// TwinCAT 3 PLC project Untitled1
// ProgramVersion: 3.1.4023.0
// libraries:
//   Tc2_Standard, * (Beckhoff Automation GmbH)
//   Tc2_System, * (Beckhoff Automation GmbH)
//   Tc2_Utilities, * (Beckhoff Automation GmbH)
//   Tc3_Module, * (Beckhoff Automation GmbH)
// project tree:
//   DUTs/BundleData/ Bundle.TcDUT (not stored), Interval.TcDUT (not stored), Material.TcDUT, PositionMaterials.TcDUT (not stored)
//   DUTs/Conveyors/ Conveyor.TcPOU, ConveyorLSC.TcPOU (not stored), ConveyorMode.TcDUT (not stored), ConveyorSC.TcPOU, ConveyorSC_NC.TcPOU
//   DUTs/ SectionTask.TcDUT, Surface.TcDUT
//   GVLs/ CONSTS.TcGVL
//   HARDWARE_DISTRUBUTION/ ConveyorSyncUnit.TcPOU
//   / PlcTask.TcTTO
//   POUs/Helper Functions/ BundleIsValid.TcPOU (not stored)
//   POUs/ IndexedBuffer.TcPOU, Junction.TcPOU, MAIN.TcPOU
// real-time tasks:
//   TASK PlcTask: cycle T#10ms, priority 20, ADS port 350

CONFIGURATION Untitled1
    RESOURCE PLC ON TwinCAT3
        TASK PlcTask(INTERVAL := T#10ms, PRIORITY := 20);
        PROGRAM MAIN WITH PlcTask : MAIN;
    END_RESOURCE
END_CONFIGURATION

// ---- DUTs/BundleData/Material.TcDUT
TYPE Material :
STRUCT
	code : STRING;
	width : LREAL;
	length : LREAL;
END_STRUCT
END_TYPE
(*
use this struct to keep track of where materials are
materials enter the system when pulled from their magazine/skid and exit the system when placed on the bundle or otherwise lost
*)

// ---- DUTs/SectionTask.TcDUT
{attribute 'qualified_only'}
//{attribute 'strict'}
TYPE SectionTask :
(
	IDLE,
	ALIGN,
	ACTIVE,
	DISCHARGE,
	COMPLETE,
	
	size
);
END_TYPE

// ---- DUTs/Surface.TcDUT
{attribute 'qualified_only'}
//{attribute 'strict'}
TYPE Surface :
(
	NULL_SURFACE,
	
	TOP,
	LEFT,
	RIGHT,
	BOTTOM,
	
	TOP_LEFT,
	TOP_RIGHT,
	BOTTOM_LEFT,
	BOTTOM_RIGHT,
	
	size
);
END_TYPE

// ---- GVLs/CONSTS.TcGVL
{attribute 'qualified_only'}
VAR_GLOBAL CONSTANT
	maxQueue : DINT := 64;
	maxPairs : DINT := 16;
	
	numConveyorLines : INT := 6;
	numBuffers : INT := 20;
END_VAR

// ---- POUs/MAIN.TcPOU
PROGRAM MAIN
VAR_OUTPUT
	localTime : TIMESTRUCT;
END_VAR
VAR
	execute AT %I* : BOOL;
	trigger : R_TRIG;
	
	newBundle AT %M* : Bundle;
	newBundleConveyorsOccupied : ARRAY[1..6] OF BOOL;
	bundlesQueue : ARRAY[0..CONSTS.maxQueue] OF Bundle;
	numBundles : INT;
	
	buffers : ARRAY[1..CONSTS.numBuffers] OF IndexedBuffer;
END_VAR
VAR //transfer junctions are clear
	transferJunctionClear_A4 AT %I* : BOOL;
	transferJunctionClear_A5 AT %I* : BOOL;
	transferJunctionClear_A2 AT %I* : BOOL;
END_VAR
VAR CONSTANT //area 3 indexes for the transfer junctions
	transferJunctionIndex_A4 : INT := 5;
	transferJunctionIndex_A5 : INT := 10;
	transferJunctionIndex_A2 : INT := 20;
END_VAR

(*
Area 3 contains <n> buffers, each index contains 6 conveyors
	this allows each buffer to carry up to a theoretical maximum of 6 bundles - realistically this will be limited to 3

implementation:
	each buffer stores 6 iterators (1 for each conveyor) to point to an element in bundlesQueue, and a master conveyor mode request
	set the requested mode for all conveyors within a buffer to the highest priority request
	then use an external module calculate the links and set the modes
	
on receipt of new bundle:
	add to bundle queue
	identify which conveyor lines the bundle sits on
*)

initialize();
callBuffers();

METHOD PRIVATE blocks : BOOL
VAR_INPUT
END_VAR
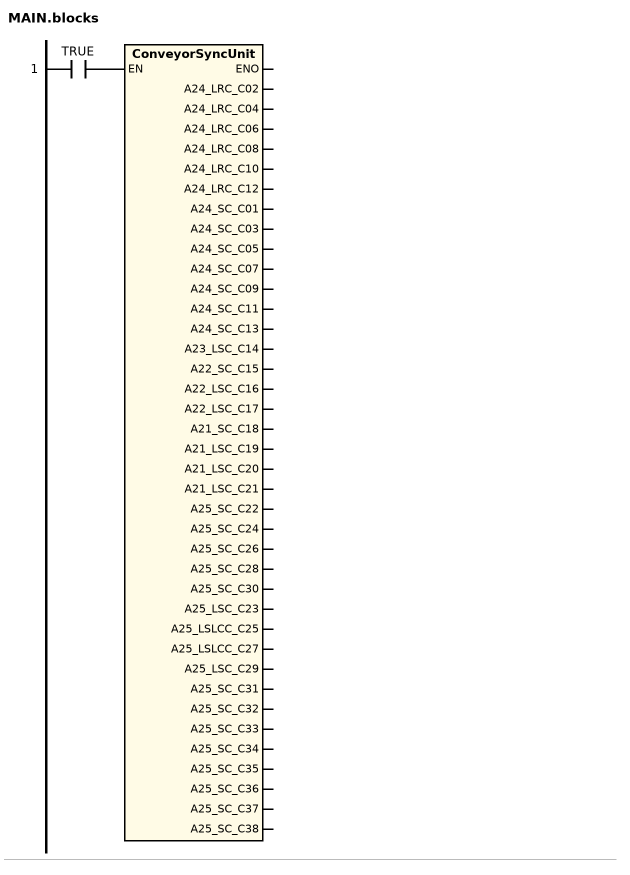
// NETWORK 1
ConveyorSyncUnit();
END_METHOD

METHOD callBuffers : BOOL
VAR_INPUT
END_VAR
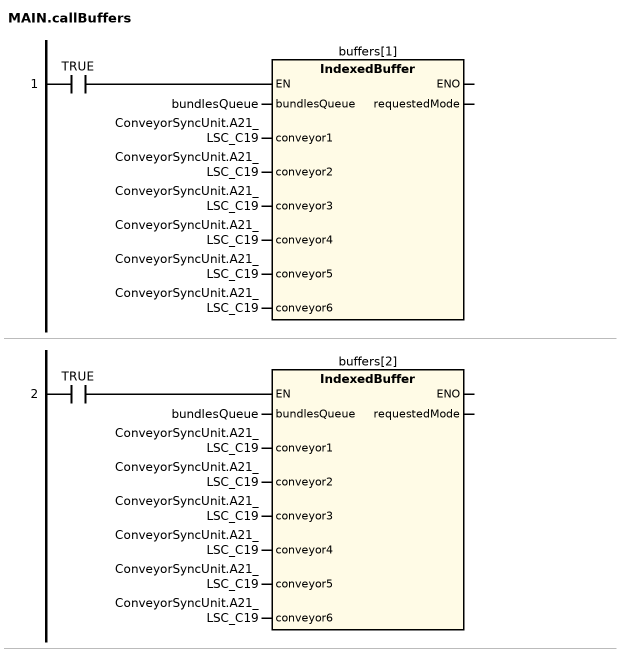
// NETWORK 1
buffers[1](
    bundlesQueue := bundlesQueue,
    conveyor1 := ConveyorSyncUnit.A21_LSC_C19,
    conveyor2 := ConveyorSyncUnit.A21_LSC_C19,
    conveyor3 := ConveyorSyncUnit.A21_LSC_C19,
    conveyor4 := ConveyorSyncUnit.A21_LSC_C19,
    conveyor5 := ConveyorSyncUnit.A21_LSC_C19,
    conveyor6 := ConveyorSyncUnit.A21_LSC_C19); // IndexedBuffer

// NETWORK 2
buffers[2](
    bundlesQueue := bundlesQueue,
    conveyor1 := ConveyorSyncUnit.A21_LSC_C19,
    conveyor2 := ConveyorSyncUnit.A21_LSC_C19,
    conveyor3 := ConveyorSyncUnit.A21_LSC_C19,
    conveyor4 := ConveyorSyncUnit.A21_LSC_C19,
    conveyor5 := ConveyorSyncUnit.A21_LSC_C19,
    conveyor6 := ConveyorSyncUnit.A21_LSC_C19); // IndexedBuffer
END_METHOD

METHOD PRIVATE handleJunctions : BOOL
VAR_INPUT
END_VAR
(*
special junction indexes (temporary):
	A4: 5
	A5: 10
	A2: 20
*)

(*
if junction is occupied:
	conveyor before junction cannot move FWD
	conveyor after junction cannot move BCK
	
consecutive occupied conveyors must be chained to the same motion
	use ConveyorSyncUnit PRG
*)
END_METHOD

METHOD PRIVATE initialize : BOOL
VAR
	i : INT;
END_VAR
FOR i:=1 TO CONSTS.numBuffers-1 BY 1 DO
	buffers[i].connectTo(next:= ADR(buffers[i+1]));
END_FOR
END_METHOD

METHOD PRIVATE receive : BOOL
VAR
	i : DINT;
END_VAR
FOR i:=0 TO CONSTS.maxQueue BY 1 DO
	
	IF NOT BundleIsValid(bundlesQueue[i]) THEN
		bundlesQueue[i] := newBundle;
		
		receive := TRUE;
		EXIT;
	END_IF
	
END_FOR

//read newBundleConveyorsOccupied[] to see which conveyor lines the bundle sits on
END_METHOD

END_PROGRAM

// ---- POUs/IndexedBuffer.TcPOU
FUNCTION_BLOCK IndexedBuffer
VAR_IN_OUT
	bundlesQueue : ARRAY[*] OF Bundle;
	
	conveyor1 : ConveyorSC; //left/outer
	conveyor2 : ConveyorSC;
	conveyor3 : ConveyorSC;
	conveyor4 : ConveyorSC;
	conveyor5 : ConveyorSC;
	conveyor6 : ConveyorSC; //right/inner
END_VAR
VAR_OUTPUT
	requestedMode : ConveyorMode;
	trueMode : ConveyorMode;
END_VAR
VAR
	nextBuffer : POINTER TO IndexedBuffer; //no next buffer = junction*
	prevBuffer : POINTER TO IndexedBuffer;
	
	conveyors : ARRAY[1..CONSTS.numConveyorLines] OF POINTER TO ConveyorSC;
	iBundles : ARRAY[1..CONSTS.numConveyorLines] OF INT := [6(-1)];
	
	step : SectionTask;
END_VAR
VAR
	i : INT;
END_VAR

(*
this FB represents an indexed buffer for area 3
up to 6 bundles per buffer, 1 per conveyor line
	assumes 6 independent conveyer drivers
*)

fillConveyorsArray();
setConveyorMode();

(*
each section will read and copy the iterators from the previous buffer when ready
	buffers cannot write their iterators to the next buffer as the next buffer may still be active
*)

CASE step OF
	SectionTask.IDLE:
		requestedMode := ConveyorMode.IDLE;
	
		IF prevBuffer <> 0 THEN //if has previous buffer, get the iterators from there
			step := SEL(prevBuffer^.iteratorsAreValid(), 0, SectionTask.ALIGN);
			(*
			IF prevBuffer^.iteratorsAreValid() THEN
				step := SectionTask.ALIGN;
			END_IF
			*)
		ELSIF iteratorsAreValid() THEN //this is the first buffer - conveyor-bundle iterators should be assigned via receiveNewIndexes()
			step := SectionTask.DISCHARGE; //since bundles are already on the buffer, next step should be discharge
			
		END_IF
	(*
	SectionTask.ACTIVE:
		CASE masterConveyorTrueMode OF
			
		END_CASE
	*)
	SectionTask.ALIGN:
		requestedMode := ConveyorMode.FORWARD;
		
		IF NOT allConveyorsVacant() THEN //at least 1 conveyor is occupied
			iBundles := SEL(prevBuffer <> 0, iBundles, prevBuffer^.iBundles);
			step := SectionTask.DISCHARGE;
		END_IF
		
	SectionTask.ACTIVE: //
	
	SectionTask.DISCHARGE:		
		IF nextBuffer <> 0 THEN
			requestedMode := ConveyorMode.FORWARD;
			
			IF allConveyorsVacant() THEN //all conveyors vacant
				step := SectionTask.COMPLETE;
			END_IF
			
		ELSE //no next buffer - upcoming junction
			(*
			0 - set all conveyors to stop
			1 - stop conveyors at exit sensor
			2 - identify the conveyors which carry bundles that do not need transfer
				move those conveyors forward
				set their respective bundle iterators to 0 when vacant
				remaining occupied conveyors carry bundles that require transfer
			3 - transfer the remaining bundles in order of lowest index
				
			*)
			
		END_IF
		
		
	SectionTask.COMPLETE:
		requestedMode := ConveyorMode.IDLE;
		
		resetIterators();
		step := 0;
		
END_CASE

METHOD PROTECTED allConveyorsOccupied : BOOL
VAR_INPUT
END_VAR
VAR
	i : INT;
END_VAR
FOR i:=1 TO CONSTS.numConveyorLines BY 1 DO
	IF NOT conveyors[i]^.IsOccupied THEN
		RETURN;
	END_IF
END_FOR

allConveyorsOccupied := TRUE;
END_METHOD

METHOD PROTECTED allConveyorsVacant : BOOL
VAR_INPUT
END_VAR
VAR
	i : INT;
END_VAR
FOR i:=1 TO CONSTS.numConveyorLines BY 1 DO
	IF conveyors[i]^.IsOccupied THEN
		RETURN;
	END_IF
END_FOR

allConveyorsVacant := TRUE;
END_METHOD

METHOD PROTECTED computeLinks : BOOL
VAR_OUTPUT
	priorityRequest : ConveyorMode;
	trueMode : ConveyorMode;
END_VAR
VAR
	i : INT;
END_VAR
FOR i:=1 TO CONSTS.numConveyorLines BY 1 DO //calculate the highest priority request
	priorityRequest := MAX(priorityRequest, conveyors[i]^.requestedMode);
END_FOR

FOR i:=1 TO CONSTS.numConveyorLines BY 1 DO //set all conveyors to that highest priority request
	conveyors[i]^.setRequest(newRequest:= priorityRequest);
END_FOR
END_METHOD

METHOD connectTo : BOOL
VAR_INPUT
	next : POINTER TO IndexedBuffer;
END_VAR
nextBuffer := next;

IF next <> 0 THEN
	next^.prevBuffer := THIS;
END_IF
END_METHOD

METHOD conveyorsAtSensorExit : BOOL
VAR
	i : INT;
END_VAR
FOR i:=1 TO CONSTS.numConveyorLines BY 1 DO
	IF iBundles[i] <> -1 THEN
		
		RETURN;
	END_IF
END_FOR

conveyorsAtSensorExit := TRUE;
END_METHOD

METHOD PROTECTED fillConveyorsArray : BOOL
VAR_INPUT
END_VAR
{warning disable C0371}
conveyors[1] := ADR(conveyor1);
conveyors[2] := ADR(conveyor2);
conveyors[3] := ADR(conveyor3);
conveyors[4] := ADR(conveyor4);
conveyors[5] := ADR(conveyor5);
conveyors[6] := ADR(conveyor6);
END_METHOD

METHOD PROTECTED iteratorsAreValid : BOOL
VAR
	i : INT;
END_VAR
FOR i:=1 TO CONSTS.numConveyorLines BY 1 DO
	IF iBundles[i] <> -1 THEN
		iteratorsAreValid := TRUE;
		RETURN;
	END_IF
END_FOR
END_METHOD

METHOD receiveNewIterators : BOOL
VAR_INPUT
	iLine1 : INT;
	iLine2 : INT;
	iLine3 : INT;
	iLine4 : INT;
	iLine5 : INT;
	iLine6 : INT;
END_VAR
//6 ints containing the new array indexes of the new bundles in bundlesQueue, 1 for each respective conveyor line
//-1 indicates unused, non-negative are real indexes
iBundles[1] := iLine1;
iBundles[2] := iLine1;
iBundles[3] := iLine1;
iBundles[4] := iLine1;
iBundles[5] := iLine1;
iBundles[6] := iLine1;
END_METHOD

METHOD PROTECTED resetIterators : BOOL
VAR_INPUT
END_VAR
VAR
	i : INT;
END_VAR
FOR i:=1 TO CONSTS.numConveyorLines BY 1 DO
	iBundles[i] := -1;
END_FOR
END_METHOD

METHOD PROTECTED setConveyorMode : BOOL
VAR
	i : INT;
END_VAR
FOR i:=1 TO CONSTS.numConveyorLines BY 1 DO
	conveyors[i]^.setRequest(newRequest:= requestedMode);
END_FOR

FOR i:=1 TO CONSTS.numConveyorLines BY 1 DO
	trueMode := MAX(trueMode, conveyors[i]^.trueMode);
END_FOR
END_METHOD

END_FUNCTION_BLOCK

// ---- DUTs/Conveyors/ConveyorSC.TcPOU
FUNCTION_BLOCK ConveyorSC
VAR_INPUT
	bEnable : BOOL;
END_VAR
VAR_OUTPUT
	trueMode : ConveyorMode;
	requestedMode : ConveyorMode;
	
	error AT %I* : BOOL;
	position AT %I* : REAL;
	velocity AT %I* : REAL;
	
	sensorEntry AT %I* : BOOL := TRUE;
	sensorExit AT %I* : BOOL;
END_VAR
VAR
	enable AT %Q* : BOOL := TRUE;
	direction AT %Q* : BOOL; //FALSE = forward, TRUE = backward
	pulse AT %Q* : BOOL;
	reset AT %Q* : BOOL;	
END_VAR
VAR
	//nextConveyor : POINTER TO ConveyorSC;
	//prevConveyor : POINTER TO ConveyorSC;
	
	pulser : TP; //pulses are assumed to be low-high-low
END_VAR
VAR_STAT CONSTANT
	pulseWidth : TIME := T#50MS;
END_VAR
(*
standard slat conveyor - no lifter
compliant with PLCopen motion control
*)

enable := bEnable;

override();

sequence();

METHOD backward : BOOL
VAR_INPUT
END_VAR
END_METHOD

METHOD forward : BOOL
VAR_INPUT
END_VAR
END_METHOD

{attribute 'monitoring' := 'call'}
PROPERTY IsOccupied : BOOL
GET
IsOccupied := sensorExit OR sensorEntry;
END_GET
END_PROPERTY

METHOD join : BOOL
VAR_INPUT
	conveyor : POINTER TO ConveyorSC;
END_VAR
//nextConveyor := conveyor;
//conveyor^.prevConveyor := THIS;
END_METHOD

METHOD PROTECTED override : BOOL
VAR_INPUT
END_VAR
END_METHOD

METHOD reset : BOOL
VAR_INPUT
END_VAR
position := 0;
velocity := velocity; //no change
END_METHOD

METHOD PROTECTED sequence : BOOL
VAR_INPUT
END_VAR
direction := (trueMode = ConveyorMode.BACKWARD); //set direction bit

pulser(IN:= , PT:= pulseWidth, Q=> pulse, ET=> );
pulser.IN := 
	enable AND 
	NOT error AND 
	NOT reset AND 
	(trueMode = ConveyorMode.FORWARD OR trueMode = ConveyorMode.BACKWARD)
	AND pulser.Q; //ends pulse itself
END_METHOD

METHOD setMode : BOOL
VAR_INPUT
	mode : ConveyorMode;
END_VAR
trueMode := mode;
END_METHOD

METHOD setRequest : BOOL
VAR_INPUT
	newRequest : ConveyorMode;
END_VAR
requestedMode := newRequest;
END_METHOD

METHOD target : BOOL
VAR_INPUT
	targetPosition : REAL;
END_VAR
END_METHOD

END_FUNCTION_BLOCK

// ---- DUTs/Conveyors/Conveyor.TcPOU
FUNCTION_BLOCK Conveyor
VAR_INPUT
	bEnable : BOOL;
END_VAR
VAR_OUTPUT	
	enable AT %Q* : BOOL;
	direction AT %Q* : BOOL; //FALSE = forward, TRUE = backward
	pulse AT %Q* : BOOL;
	reset AT %Q* : BOOL;
	
	error AT %I* : BOOL;
	sensorEntry AT %I* : BOOL;
	sensorExit AT %I* : BOOL;
	
	//vertical conveyors only
	requestLifter: BOOL;

	lifterEnable AT %Q* : BOOL := TRUE;
	lifterDirection AT %Q* : BOOL; //FALSE = up, TRUE = down
	lifterPulse AT %Q* : BOOL;
	lifterReset AT %Q* : BOOL;
	
	lifterError AT %I* : BOOL;
	extended AT %I* : BOOL;
	retracted AT %I* : BOOL;
END_VAR
VAR_OUTPUT
	position AT %I* : REAL;
	velocity AT %I* : REAL;
END_VAR
VAR
	operation : ConveyorMode;
	request : ConveyorMode;
	
	//pulses are assumed to be low-HIGH-low
	pulser : TP;
	lifterPulser : TP;
	
	hasLifter : BOOL;
END_VAR
VAR_STAT CONSTANT
	pulseWidth : TIME := T#25MS;
END_VAR

pulser(IN:= , PT:= pulseWidth, Q=> pulse, ET=> );

direction := (operation = ConveyorMode.BACKWARD);

pulser.IN := 
	enable AND 
	NOT error AND 
	NOT reset AND 
	(operation = ConveyorMode.FORWARD OR operation = ConveyorMode.BACKWARD);

IF pulser.IN AND NOT pulser.Q THEN
	pulser.IN := FALSE;
END_IF

lifterPulser(IN:= , PT:= pulseWidth, Q=> lifterPulse, ET=> );

lifterPulser.IN := 
	hasLifter AND
	lifterEnable AND 
	NOT lifterError AND 
	NOT lifterReset AND 
	requestLifter;
	
IF lifterPulser.IN AND NOT lifterPulser.Q THEN
	lifterPulser.IN := FALSE;
END_IF

METHOD backward : BOOL
VAR_INPUT
END_VAR
END_METHOD

METHOD extend : BOOL
VAR_INPUT
END_VAR
END_METHOD

METHOD forward : BOOL
VAR_INPUT
END_VAR
END_METHOD

METHOD occupied : BOOL
occupied := sensorExit OR sensorEntry;
END_METHOD

METHOD reset : BOOL
VAR_INPUT
END_VAR
position := 0;
velocity := velocity; //no change

extend();
END_METHOD

METHOD retract : BOOL
VAR_INPUT
END_VAR
END_METHOD

METHOD setOperation : BOOL
VAR_INPUT
	newOperation : ConveyorMode;
END_VAR
operation := newOperation;
END_METHOD

METHOD setRequest : BOOL
VAR_INPUT
	requestedMode : ConveyorMode;
END_VAR
request := requestedMode;
END_METHOD

METHOD target : BOOL
VAR_INPUT
	targetPosition : REAL;
END_VAR
END_METHOD

END_FUNCTION_BLOCK

// ---- HARDWARE_DISTRUBUTION/ConveyorSyncUnit.TcPOU
PROGRAM ConveyorSyncUnit
(*
this module was copied over from Area2v2a
must be modified to link IndexedBuffers, not individual conveyors
*)
VAR_OUTPUT	
	A24_LRC_C02 	: Conveyor; //these conveyoors move bundles from A2.7 to A2.4
	A24_LRC_C04 	: Conveyor;
	A24_LRC_C06	 	: Conveyor;
	A24_LRC_C08 	: Conveyor;
	A24_LRC_C10 	: Conveyor;
	A24_LRC_C12 	: Conveyor;
	
	A24_SC_C01 		: ConveyorSC; //these conveyors move bundles on A2.4 forward down the cell
	A24_SC_C03 		: ConveyorSC;
	A24_SC_C05 		: ConveyorSC;
	A24_SC_C07 		: ConveyorSC;
	A24_SC_C09 		: ConveyorSC;
	A24_SC_C11 		: ConveyorSC;
	A24_SC_C13 		: ConveyorSC;
	
	A23_LSC_C14 	: ConveyorLSC;
	
	A22_SC_C15 		: ConveyorSC;
	A22_LSC_C16 	: ConveyorLSC;
	A22_LSC_C17 	: ConveyorLSC;
	
	A21_SC_C18 		: ConveyorSC;
	A21_LSC_C19 	: ConveyorLSC;
	A21_LSC_C20 	: ConveyorLSC;
	A21_LSC_C21 	: ConveyorLSC;
	
	A25_SC_C22 		: ConveyorSC;
	A25_SC_C24 		: ConveyorSC;
	A25_SC_C26 		: ConveyorSC;
	A25_SC_C28 		: ConveyorSC;
	A25_SC_C30 		: ConveyorSC;
	
	A25_LSC_C23 	: ConveyorLSC; //these conveyors move the bundle sideways onto the output buffers
	A25_LSLCC_C25 	: ConveyorLSC;
	A25_LSLCC_C27 	: ConveyorLSC;
	A25_LSC_C29 	: ConveyorLSC;
	A25_SC_C31 		: ConveyorSC;
	A25_SC_C32 		: ConveyorSC;
	A25_SC_C33 		: ConveyorSC;
	A25_SC_C34 		: ConveyorSC;
	A25_SC_C35 		: ConveyorSC;
	A25_SC_C36 		: ConveyorSC;
	A25_SC_C37 		: ConveyorSC;
	A25_SC_C38 		: ConveyorSC;
END_VAR
VAR
	cellConveyors : ARRAY[1..numCellConveyors] OF POINTER TO ConveyorSC;
	receiverConveyors : ARRAY[1..numReceiverConveyors] OF POINTER TO ConveyorSC;
	outputConveyors : ARRAY[1..numOutputConveyors] OF POINTER TO ConveyorSC;
	
	spoolTimer : TON;
	i : DINT := 1;
END_VAR
VAR CONSTANT
	spoolSpacing : TIME := T#100MS;
	
	numTotalConveyors : INT := 38;
	
	numCellConveyors : INT := 20;
	
	numReceiverConveyors : INT := 6;
	numOutputConveyors : INT := 12;
END_VAR
(*
this module contains all conveyors to be distributed to subareas as needed
by not tying conveyors to any particular subarea, any subarea will have some access to any conveyor
*)

fillCellConveyors();
fillOutputConveyors();

computeCellLinks();

spoolTimer(IN:= , PT:= spoolSpacing, Q=> , ET=> );
spoolTimer.IN := TRUE;

IF
	( //conveyor requests motion
		cellConveyors[i]^.requestedMode = ConveyorMode.FORWARD OR 
		cellConveyors[i]^.requestedMode = ConveyorMode.BACKWARD
	) AND
	cellConveyors[i]^.requestedMode <> cellConveyors[i]^.trueMode AND //conveyor request differs from current mode
	spoolTimer.Q //ready to spool
THEN
	//spool up conveyor
	i := (i + 1) MOD (numCellConveyors + 1) + 1;
	spoolTimer.IN := FALSE;
END_IF

METHOD PRIVATE computeCellLinks : BOOL
VAR
	i : DINT;
	j : DINT;
	
	linkStart : DINT := -1;
	linkEnd : DINT := -1;
	
	priorityInLink : ConveyorMode;
END_VAR
(*
link interation method 
will correctly set all operations every cycle
*)
FOR i:=1 TO numCellConveyors BY 1 DO
	IF cellConveyors[i]^.IsOccupied THEN
		
		IF linkStart = -1 THEN
			linkStart := i;
		END_IF
		
		priorityInLink := MAX(priorityInLink, cellConveyors[i]^.requestedMode);
		linkEnd := i;
		
	ELSIF linkStart <> -1 AND linkEnd <> -1 THEN //set all conveyor operations to priorityInLink
		linkEnd := i-1;
		
		FOR j:=linkStart TO linkEnd BY 1 DO
			cellConveyors[j]^.setMode(priorityInLink);
		END_FOR
		
		linkStart := -1;
		linkEnd := -1;
		priorityInLink := ConveyorMode.IDLE;
		
		CONTINUE;
	END_IF
	
END_FOR


//final link
IF linkStart > -1 AND linkEnd > -1 THEN
	FOR j:=linkStart TO linkEnd BY 1 DO
		cellConveyors[j]^.setMode(priorityInLink);
	END_FOR
END_IF
END_METHOD

METHOD PRIVATE fillCellConveyors : BOOL
{warning disable C0371}
cellConveyors[1] := ADR(A24_SC_C01);
cellConveyors[2] := ADR(A24_SC_C03);
cellConveyors[3] := ADR(A24_SC_C05);
cellConveyors[4] := ADR(A24_SC_C07);
cellConveyors[5] := ADR(A24_SC_C09);
cellConveyors[6] := ADR(A24_SC_C11);
cellConveyors[7] := ADR(A24_SC_C13);

cellConveyors[8] := ADR(A23_LSC_C14);

cellConveyors[9] := ADR(A22_SC_C15);
cellConveyors[10] := ADR(A22_LSC_C16);
cellConveyors[11] := ADR(A22_LSC_C17);

cellConveyors[12] := ADR(A21_SC_C18);
cellConveyors[13] := ADR(A21_LSC_C19);
cellConveyors[14] := ADR(A21_LSC_C20);
cellConveyors[15] := ADR(A21_LSC_C21);

cellConveyors[16] := ADR(A25_SC_C22);
cellConveyors[17] := ADR(A25_SC_C24);
cellConveyors[18] := ADR(A25_SC_C26);
cellConveyors[19] := ADR(A25_SC_C28);
cellConveyors[20] := ADR(A25_SC_C30);
END_METHOD

METHOD PRIVATE fillOutputConveyors : BOOL
VAR_INPUT
END_VAR
outputConveyors[1] := ADR(A25_LSC_C23);
outputConveyors[2] := ADR(A25_LSLCC_C25);
outputConveyors[3] := ADR(A25_LSLCC_C27);
outputConveyors[4] := ADR(A25_LSC_C29);
outputConveyors[5] := ADR(A25_SC_C31);
outputConveyors[6] := ADR(A25_SC_C32);
outputConveyors[7] := ADR(A25_SC_C33);
outputConveyors[8] := ADR(A25_SC_C34);
outputConveyors[9] := ADR(A25_SC_C35);
outputConveyors[10] := ADR(A25_SC_C36);
outputConveyors[11] := ADR(A25_SC_C37);
outputConveyors[12] := ADR(A25_SC_C38);
END_METHOD

END_PROGRAM

// ---- DUTs/Conveyors/ConveyorSC_NC.TcPOU
FUNCTION_BLOCK ConveyorSC_NC
VAR_INPUT
	bEnable : BOOL;
END_VAR
VAR_OUTPUT
	sensorEntry AT %I* : BOOL := TRUE;
	sensorExit AT %I* : BOOL := TRUE;
	
	trueMode : ConveyorMode;
	requestedMode : ConveyorMode;
	
	position : LREAL;
	velocity : LREAL;
	ready : BOOL;
END_VAR
VAR
	axis : AXIS_REF;
	
	mcReadPosition : MC_ReadActualPosition; //continuous enable FBs
	mcReadVelocity : MC_ReadActualVelocity;
	mcReadError : MC_ReadAxisError;
	mcPower : MC_Power;
	
	mcReset : MC_Reset; //rising edge FBs
	mcMoveAbsolute : MC_MoveAbsolute;
	mcMoveRelative : MC_MoveRelative;
	mcMoveVelocity : MC_MoveVelocity;
	
	mcSetPosition : MC_SetPosition;
	mcStop : MC_Stop;
END_VAR
VAR_STAT CONSTANT
	targetingVelocity : INT := 500;
	continuousVelocity : INT := 500;
END_VAR
(*
this FB represents a standard slat conveyor with no lifter
	compliant with PLCopen motion control

unlike standalone servos,
	conveyors need to coordinate (not slave) their motion with other conveyors
	and be able to set their current position to any value as required by the system
	
moveAbsolute is provided for now but should not be used for position targetting and may be protected/privated later
instead, request/set the operation mode and the motion will follow
*)

IF error THEN
	stop();
	reset();
	
ELSE
	CASE trueMode OF
		ConveyorMode.IDLE:			stop();	
		ConveyorMode.FORWARD:		moveContinuous(direction:= MC_Positive_Direction);
		ConveyorMode.BACKWARD:		moveContinuous(direction:= MC_Negative_Direction);
		ConveyorMode.STOP:			stop();
	END_CASE
	
END_IF

blocks();

mcReset.Execute := FALSE;
mcMoveAbsolute.Execute := FALSE;
mcMoveRelative.Execute := FALSE;
mcMoveVelocity.Execute := FALSE;
mcSetPosition.Execute := FALSE;
mcStop.Execute := FALSE;

blocks();

PROPERTY Active : BOOL
GET
Active := 
	mcMoveAbsolute.Busy OR 
	mcMoveRelative.Busy OR 
	mcMoveVelocity.Busy OR 
	mcSetPosition.Busy OR 
	mcReset.Busy OR 
	mcStop.Busy;
END_GET
END_PROPERTY

METHOD PRIVATE blocks : BOOL
mcReadPosition(
	Axis:= axis, 
	Enable:= TRUE, 
	Valid=> , 
	Busy=> , 
	Error=> , 
	ErrorID=> , 
	Position=> position);
	
mcReadVelocity(
	Axis:= axis, 
	Enable:= TRUE, 
	Valid=> , 
	Busy=> , 
	Error=> , 
	ErrorID=> , 
	ActualVelocity=> velocity);
	
mcReadError(
	Axis:= axis, 
	Enable:= TRUE, 
	Valid=> , 
	Busy=> , 
	Error=> , 
	ErrorID=> , 
	AxisErrorID=> );
	
mcPower(
	Axis:= axis, 
	Enable:= bEnable, 
	Enable_Positive:= TRUE, 
	Enable_Negative:= TRUE, 
	Override:= 100, 
	BufferMode:= , 
	Options:= , 
	Status=> , 
	Busy=> , 
	Active=> , 
	Error=> , 
	ErrorID=> );

mcReset(
	Axis:= axis, 
	Execute:= , 
	Done=> , 
	Busy=> , 
	Error=> , 
	ErrorID=> );

mcMoveAbsolute(
	Axis:= axis, 
	Execute:= , 
	Position:= , 
	Velocity:= targetingVelocity, 
	Acceleration:= , 
	Deceleration:= , 
	Jerk:= , 
	BufferMode:= , 
	Options:= , 
	Done=> , 
	Busy=> , 
	Active=> , 
	CommandAborted=> , 
	Error=> , 
	ErrorID=> );
	
mcMoveRelative(
	Axis:= axis, 
	Execute:= , 
	Distance:= ,
	Velocity:= targetingVelocity, 
	Acceleration:= , 
	Deceleration:= , 
	Jerk:= , 
	BufferMode:= , 
	Options:= , 
	Done=> , 
	Busy=> , 
	Active=> , 
	CommandAborted=> , 
	Error=> , 
	ErrorID=> );
	
mcMoveVelocity( //stopped with stop();
	Axis:= axis, 
	Execute:= , 
	Velocity:= continuousVelocity, 
	Acceleration:= , 
	Deceleration:= , 
	Jerk:= , 
	Direction:= , 
	BufferMode:= , 
	Options:= , 
	InVelocity=> , 
	Busy=> , 
	Active=> , 
	CommandAborted=> , 
	Error=> , 
	ErrorID=> );
	
mcSetPosition(
	Axis:= axis, 
	Execute:= , 
	Position:= , 
	Mode:= , 
	Options:= , 
	Done=> , 
	Busy=> , 
	Error=> , 
	ErrorID=> );
	
mcStop(
	Axis:= axis, 
	Execute:= , 
	Deceleration:= , 
	Jerk:= , 
	Options:= , 
	Done=> , 
	Busy=> , 
	Active=> , 
	CommandAborted=> , 
	Error=> , 
	ErrorID=> );
END_METHOD

PROPERTY CurrentPosition : LREAL
GET
CurrentPosition := position;
END_GET
SET
position := CurrentPosition;
END_SET
END_PROPERTY

PROPERTY Error : BOOL
GET
error := 
	mcMoveAbsolute.Error OR 
	mcMoveRelative.Error OR 
	mcMoveVelocity.Error OR 
	mcSetPosition.Error OR 
	mcReset.Error OR 
	mcStop.Error OR
	mcReadError.AxisErrorID > 0;
END_GET
END_PROPERTY

{attribute 'monitoring' := 'call'}
PROPERTY IsOccupied : BOOL
GET
IsOccupied := sensorExit OR sensorEntry;
END_GET
END_PROPERTY

METHOD moveAbsolute : BOOL
VAR_INPUT
	newTarget : REAL;
END_VAR
mcMoveAbsolute.Position := newTarget;

IF NOT Active AND NOT error THEN
	mcMoveAbsolute.Execute := TRUE;
END_IF

moveAbsolute := 
	//mcMoveAbsolute.Done;
	CurrentPosition = TargetPosition;
END_METHOD

METHOD moveContinuous : BOOL
VAR_INPUT
	direction : MC_Direction;
END_VAR
mcMoveVelocity.Direction := direction;

IF NOT Active AND NOT error THEN
	mcMoveVelocity.Execute := TRUE;
	moveContinuous := TRUE;
END_IF
END_METHOD

METHOD reset : BOOL
VAR_INPUT
END_VAR
mcReset.Execute := TRUE;

reset := mcReset.Done;
END_METHOD

METHOD setMode : BOOL
VAR_INPUT
	mode : ConveyorMode;
END_VAR
trueMode := mode;
END_METHOD

METHOD setRequest : BOOL
VAR_INPUT
	newRequest : ConveyorMode;
END_VAR
requestedMode := newRequest;
END_METHOD

METHOD stop : BOOL
VAR_INPUT
END_VAR
mcStop.Execute := TRUE;

mcMoveAbsolute.Execute := FALSE;
mcMoveRelative.Execute := FALSE;
mcMoveVelocity.Execute := FALSE;
END_METHOD

PROPERTY TargetPosition : LREAL
GET
END_GET
SET
moveAbsolute(newTarget := TargetPosition);
END_SET
END_PROPERTY

END_FUNCTION_BLOCK

// ---- POUs/Junction.TcPOU
FUNCTION_BLOCK Junction
VAR_IN_OUT
	conveyor1 : ConveyorLSC;
	conveyor2 : ConveyorLSC;
	conveyor3 : ConveyorLSC;
	conveyor4 : ConveyorLSC;
	conveyor5 : ConveyorLSC;
	conveyor6 : ConveyorLSC;
END_VAR
VAR
	nextBuffer : POINTER TO IndexedBuffer;
	prevBuffer : POINTER TO IndexedBuffer;
	
	conveyors : ARRAY[1..CONSTS.numConveyorLines] OF POINTER TO ConveyorSC;
	iBundles : ARRAY[1..CONSTS.numConveyorLines] OF INT := [6(-1)];
	
	step : SectionTask;
END_VAR

CASE step OF
	SectionTask.IDLE:
		
		
	SectionTask.ALIGN:
		
		
	SectionTask.ACTIVE:
		(*
		1	send all bundles that do no need area transfer over the junction 
			-iterate through array of iterators
				*if bundle does not need transfer then request the conveyor FWD
				*if bundle needs transfer, then hold the conveyor
			
		2	 
		*)
	
	
END_CASE

END_FUNCTION_BLOCK
